ABB RAPID module: MainModule.MOD

MODULE MainModule
	CONST robtarget home:=[[-12.71,280.55,565.13],[1.27104E-05,0.999859,0.0168188,-2.49647E-06],[1,0,-1,0],[9E+09,9E+09,9E+09,9E+09,9E+09,9E+09]];
	CONST robtarget ql:=[[546.75,-68.63,212.08],[0.0164627,0.619264,0.784759,0.019849],[-1,0,-4,0],[9E+09,9E+09,9E+09,9E+09,9E+09,9E+09]];
	CONST robtarget sj:=[[-45.41,426.33,467.16],[0.00404631,0.946945,0.320535,0.0231567],[1,-1,-2,0],[9E+09,9E+09,9E+09,9E+09,9E+09,9E+09]];
	CONST robtarget fl:=[[470.89,200.38,291.53],[0.00349261,0.940841,0.337883,0.0253256],[0,-1,-3,0],[9E+09,9E+09,9E+09,9E+09,9E+09,9E+09]];
	CONST robtarget ls{2}:=[[[310.51,221.34,280.80],[0.00417547,0.946907,0.320621,0.0235096],[0,-1,-3,0],[9E+09,9E+09,9E+09,9E+09,9E+09,9E+09]],[[346.76,221.69,282.01],[0.00416857,0.94692,0.320581,0.0235366],[0,-1,-3,0],[9E+09,9E+09,9E+09,9E+09,9E+09,9E+09]]];
	CONST robtarget lsk:=[[11.97,278.75,292.92],[0.00407899,0.946941,0.320532,0.0233428],[0,-1,-2,0],[9E+09,9E+09,9E+09,9E+09,9E+09,9E+09]];
	CONST robtarget fwl:=[[-231.77,253.16,290.26],[0.0119305,-0.940746,-0.338457,-0.0173771],[1,-1,-1,0],[9E+09,9E+09,9E+09,9E+09,9E+09,9E+09]];
	PROC main()
		<SMT>
	ENDPROC
ENDMODULE
